(* IEC 61131-3 sources: beckhoffAutomationInterface/ST/Shark/Lib/Hardware/Interfaces, 9 files *)

(* ---- I_AnalogOutput.st ---- *)
(* Analog output interface for hardware abstraction. *)
INTERFACE I_AnalogOutput EXTENDS I_Errorable

METHOD SetOutput
VAR_INPUT
    nValue : INT;  // Raw analog value (typically 0-32767 for 0-100%)
END_VAR
END_METHOD

METHOD SetPercentage
VAR_INPUT
    rPercentage : REAL;  // Percentage value (0.0 - 100.0)
END_VAR
END_METHOD

METHOD GetOutput : INT
END_METHOD

METHOD GetPercentage : REAL
END_METHOD

(* Apply the safe raw value configured at Init time.
   Called by behaviour-tree nodes on Halt — the node has no knowledge of
   what the safe value is for this particular output. *)
METHOD SetSafeState
END_METHOD

END_INTERFACE

(* ---- I_DigitalInput.st ---- *)
(* Digital input interface for boolean sensing. *)
INTERFACE I_DigitalInput

METHOD GetState : BOOL
END_METHOD

END_INTERFACE

(* ---- I_DigitalOutput.st ---- *)
(* Digital output interface for boolean control. *)
INTERFACE I_DigitalOutput

METHOD SetOutput
VAR_INPUT
    bValue : BOOL;
END_VAR
END_METHOD

METHOD GetOutput : BOOL
END_METHOD

(* Apply the safe state configured at Init time.
   Called by behaviour-tree nodes on Halt — the node has no knowledge of
   whether safe means TRUE or FALSE for this particular output. *)
METHOD SetSafeState
END_METHOD

END_INTERFACE

(* ---- I_HardwareProvider.st ---- *)
(* Common hardware-access surface shared across all machines that use the
   dual-sided gas-delivery pattern (PRO, Shark, future variants).

   Contains ONLY the methods whose signatures are identical across all
   participating machines:
     - Side-abstracted getters keyed on E_GasSide (a Lib enum)
     - Zero-input getters for shared singletons (mix valve, exhaust pump,
       exhaust pressure sensor, etc.)
     - All thermal getters defined directly in this interface

   Per-machine variations (enums) are passed as INT to the generic getters
   below — enum-to-INT is implicit in IEC 61131-3. This eliminates the need
   for machine-specific interface extensions (I_PROHardwareProvider, etc.).

   Gas Flow Path (per side):
     Carrier Gas → MFC/Gas Valve → CM Bubbler Inlet → Bubbler →
     HM Bubbler Outlet → Hot Manifold → PCV → Start Valve → Nozzle *)
INTERFACE I_HardwareProvider EXTENDS __System.IQueryInterface

    // =========================================================================
    // VALVE GETTERS - Side-abstracted
    // =========================================================================
METHOD GetGasIsoValve : I_Valve
VAR_INPUT
    eSide : E_GasSide;
    nBubblerIndex : DINT;
END_VAR
END_METHOD

METHOD GetCMBubblerValve : I_Valve
VAR_INPUT
    eSide : E_GasSide;
    nBubblerIndex : DINT;
END_VAR
END_METHOD

METHOD GetHMBubblerValve : I_Valve
VAR_INPUT
    eSide : E_GasSide;
    nBubblerIndex : DINT;
END_VAR
END_METHOD

METHOD GetCMPurgeValve : I_Valve
VAR_INPUT
    eSide : E_GasSide;
END_VAR
END_METHOD

METHOD GetHMPurgeValve : I_Valve
VAR_INPUT
    eSide : E_GasSide;
END_VAR
END_METHOD

METHOD GetCMVacuumIsoValve : I_Valve
VAR_INPUT
    eSide : E_GasSide;
END_VAR
END_METHOD

METHOD GetHMVacuumIsoValve : I_Valve
VAR_INPUT
    eSide : E_GasSide;
END_VAR
END_METHOD

METHOD GetNozzleIsoValve : I_Valve
VAR_INPUT
    eSide : E_GasSide;
END_VAR
END_METHOD

    // =========================================================================
    // VALVE GETTERS - Common (no side)
    // =========================================================================
METHOD GetMixValve : I_Valve
END_METHOD

METHOD GetExhaustVacuumIsoValve : I_Valve
END_METHOD

    // =========================================================================
    // DIGITAL OUTPUT GETTERS - Common
    // =========================================================================
METHOD GetExhaustPump : I_DigitalOutput
END_METHOD

    // =========================================================================
    // SENSOR GETTERS - Side-abstracted
    // =========================================================================
METHOD GetCMPressureSensor : I_Sensor
VAR_INPUT
    eSide : E_GasSide;
END_VAR
END_METHOD

METHOD GetHMPressureSensor : I_Sensor
VAR_INPUT
    eSide : E_GasSide;
END_VAR
END_METHOD

METHOD GetMFCFlowSensor : I_Sensor
VAR_INPUT
    eSide : E_GasSide;
END_VAR
END_METHOD

    // =========================================================================
    // SENSOR GETTERS - Common
    // =========================================================================
METHOD GetExhaustPressureSensor : I_Sensor
END_METHOD

    // =========================================================================
    // CONTROLLER GETTERS - Side-abstracted
    // =========================================================================
METHOD GetMFCController : I_Controller
VAR_INPUT
    eSide : E_GasSide;
END_VAR
END_METHOD

METHOD GetPressureController : I_Controller
VAR_INPUT
    eSide : E_GasSide;
END_VAR
END_METHOD

    // =========================================================================
    // CONTROLLER GETTERS - Inert Gas (used by SpotDeposition)
    // =========================================================================
METHOD GetInertMFCController : I_Controller
END_METHOD

    // =========================================================================
    // VALVE GETTERS - Inert Gas (used by SpotDeposition)
    // =========================================================================
METHOD GetInertGasValve : I_Valve
END_METHOD

    // =========================================================================
    // SUBSYSTEM GETTERS
    // =========================================================================

    // Returns the machine-specific chuck-vacuum subsystem.
    // Lib chuck-vacuum sequences depend on this abstraction to remain
    // portable across machines with different pump/valve/sensor topologies.
METHOD GetChuckVacuumSystem : I_ChuckVacuumSystem
END_METHOD

    // =========================================================================
    // GENERIC GETTERS - Index-based (pass machine enum; implicit INT cast)
    // =========================================================================
METHOD GetValve : I_Valve
VAR_INPUT
    nIndex : INT;
END_VAR
END_METHOD

METHOD GetDigitalOutput : I_DigitalOutput
VAR_INPUT
    nIndex : INT;
END_VAR
END_METHOD

METHOD GetDigitalInput : I_DigitalInput
VAR_INPUT
    nIndex : INT;
END_VAR
END_METHOD

METHOD GetPressureSensor : I_Sensor
VAR_INPUT
    nIndex : INT;
END_VAR
END_METHOD

METHOD GetFlowController : I_Controller
VAR_INPUT
    nIndex : INT;
END_VAR
END_METHOD

METHOD GetTemperatureController : I_Controller
VAR_INPUT
    nIndex : INT;
END_VAR
END_METHOD

    // Individual heater CHANNEL controller addressed by its flat global channel
    // index (1..CHANNEL_MAX). Pass the machine E_HeatChannel enum (implicit INT).
METHOD GetTemperatureChannel : I_Controller
VAR_INPUT
    nGlobalIdx : INT;
END_VAR
END_METHOD

METHOD GetPressureControllerById : I_Controller
VAR_INPUT
    nIndex : INT;
END_VAR
END_METHOD

    // =========================================================================
    // UTILITY & CONFIGURATION
    // =========================================================================
METHOD IsGasMode : BOOL
VAR_INPUT
    eSide : E_GasSide;
    nBubblerIndex : DINT;
END_VAR
END_METHOD

METHOD GetMaxBubblerCount : DINT
VAR_INPUT
    eSide : E_GasSide;
END_VAR
END_METHOD

    // =========================================================================
    // TEMPERATURE CONTROLLER GETTERS
    // =========================================================================
METHOD GetHMTemperatureController : I_Controller
VAR_INPUT
    eSide : E_GasSide;
END_VAR
END_METHOD

METHOD GetUmbilicalTemperatureController : I_Controller
VAR_INPUT
    eSide : E_GasSide;
END_VAR
END_METHOD

METHOD GetBubblerTemperatureController : I_Controller
VAR_INPUT
    eSide : E_GasSide;
    nBubblerIndex : DINT;
END_VAR
END_METHOD

METHOD GetHeadTemperatureController : I_Controller
END_METHOD

METHOD GetExhaustTemperatureController : I_Controller
END_METHOD

METHOD GetChuckTemperatureController : I_Controller
END_METHOD

END_INTERFACE

(* ---- I_LevelStage.st ---- *)
(* Adjustable level (0..100 %) stage interface.

Typically combined with I_OnOffStage on the same FB: the on/off interface
gates power; the level interface sets the analog trim. A device that only
supports on/off does NOT implement I_LevelStage, so callers cannot
accidentally request a setpoint that has no effect. *)
INTERFACE I_LevelStage

METHOD SetLevel : BOOL
VAR_INPUT
    rPercentage : REAL;
END_VAR
END_METHOD

METHOD GetLevel : REAL
END_METHOD

END_INTERFACE

(* ---- I_OnOffStage.st ---- *)
(* Generic on/off stage interface.

A device that can be enabled or disabled with no level/intensity control.
Examples: a digitally-switched ozone generator, a UV lamp, a heater fan
running at fixed speed.

Combine with I_LevelStage on the same FB if the device also accepts an
analog trim setpoint (see FB_OnOffLevelStage). *)
INTERFACE I_OnOffStage EXTENDS __System.IQueryInterface

METHOD Enable : BOOL
VAR_INPUT
    bEnable : BOOL;
END_VAR
END_METHOD

METHOD IsEnabled : BOOL
END_METHOD

METHOD Execute : BOOL
END_METHOD

END_INTERFACE

(* ---- I_RawAnalogInput.st ---- *)
(* Abstracts the raw hardware input for analog sensors.

   nRawValue is DINT so a single interface covers both 16-bit terminals
   (EL32xx RTD / EL31xx, INT sign-extended to DINT) and 32-bit terminals
   (EL3314 thermocouple, native DINT). DINT is a lossless superset of INT. *)
INTERFACE I_RawAnalogInput
METHOD GetChannelState
VAR_OUTPUT
    nRawValue   : DINT;
    bError      : BOOL;
    bUnderrange : BOOL;
    bOverrange  : BOOL;
END_VAR
END_METHOD
END_INTERFACE

(* ---- I_Sensor.st ---- *)
(* Base sensor interface for measurement and error status. *)
INTERFACE I_Sensor EXTENDS I_Errorable, __System.IQueryInterface

METHOD GetMeasurement : LREAL
END_METHOD

END_INTERFACE

(* ---- I_Valve.st ---- *)
(* Valve interface - unified control for all valve types. *)
INTERFACE I_Valve EXTENDS I_Errorable

METHOD Open : BOOL
END_METHOD

METHOD Close : BOOL
END_METHOD

METHOD IsOpen : BOOL
END_METHOD

METHOD IsClosed : BOOL
END_METHOD

METHOD Reset : BOOL
END_METHOD

END_INTERFACE
